{attribute 'OPC.UA.DA' := '1'}
FUNCTION_BLOCK EvosensLight EXTENDS LightBase
VAR_INPUT
END_VAR
VAR_OUTPUT
END_VAR
VAR
	{attribute 'OPC.UA.DA' := '0'}
	_config : EvosensLightConfig;	
	{attribute 'OPC.UA.DA' := '0'}
	_coeAccess : CoeAccess;	
	{attribute 'OPC.UA.DA' := '0'}
	_initConfigSerialCom : BOOL;	
	{attribute 'OPC.UA.DA' := '0'}
	_suffix : STRING := Const.CR_LF;
	{attribute 'OPC.UA.DA' := '0'}
	_serialCom  : SerialCom(Prefix :='', Suffix := _suffix);
	{attribute 'OPC.UA.DA' := '0'}
	_refSerialCom : REFERENCE TO SerialCom(Prefix :='', Suffix := _suffix) := _serialCom;		 
	{attribute 'OPC.UA.DA' := '0'}
	_isReceived : BOOL;
	
	{attribute 'OPC.UA.DA' := '0'}
	_deliverMessages : INT;
		
	StatusMsg : STRING(255);
	SwitchOnMsg : STRING(255);
	PowerMsg : STRING(255);
	IntensityMsg : STRING(255);	
	TemperatureMsg : STRING(255);
	LightSourcesMsg : STRING(255);
	TimeLightSourceMsg  : STRING(255);
	CustomMsg : STRING(255);
		
	{region 'Commands'}
	
	{attribute 'OPC.UA.DA' := '0'}
	_setSwitchOnCmd : BOOL;
	{attribute 'OPC.UA.DA' := '0'}
	_getSwitchOnCmd : BOOL;
	{attribute 'OPC.UA.DA' := '0'}
	_setPowerCmd : BOOL;
	{attribute 'OPC.UA.DA' := '0'}
	_getPowerCmd : BOOL;
	{attribute 'OPC.UA.DA' := '0'}
	_setIntensityCmd : BOOL;
	{attribute 'OPC.UA.DA' := '0'}
	_getIntensityCmd : BOOL;
	{attribute 'OPC.UA.DA' := '0'}
	_getTimeLightSourceCmd : BOOL;
	{attribute 'OPC.UA.DA' := '0'}
	_getLightSourcesCmd : BOOL;
	{attribute 'OPC.UA.DA' := '0'}
	_customCmd : BOOL;
	{attribute 'OPC.UA.DA' := '0'}			  		   
	_raisePropertiesCmd : BOOL;
	
	{attribute 'OPC.UA.DA' := '0'}
	_lightId : UINT; 
	{attribute 'OPC.UA.DA' := '0'}
	_switchOn : BOOL;
	{attribute 'OPC.UA.DA' := '0'}
	_setPower : LREAL;
	{attribute 'OPC.UA.DA' := '0'}
	_setIntensity : LREAL;
	{attribute 'OPC.UA.DA' := '0'}
	_cmd : STRING;	
		 
	{endregion}			
	
	{attribute 'OPC.UA.DA' := '0'}
	_initDevice : BOOL;	
	 
	{attribute 'OPC.UA.DA' := '0'}
	_lightSources : ARRAY [0..Const.PHOTOLUM_NUMBER_LIGHT_SOURCE] OF STRING(255);  
	
	{attribute 'OPC.UA.DA' := '0'}
	_itemScheduler : INT;
	{attribute 'OPC.UA.DA' := '0'}
	_itemInitScheduler : INT;
	{attribute 'OPC.UA.DA' := '0'}
	_itemExecScheduler : INT;		
	{attribute 'OPC.UA.DA' := '0'}
	_itemRaisedProperties : INT;			
	{attribute 'OPC.UA.DA' := '0'}
	_pulseGenerator : TON;	
	{attribute 'OPC.UA.DA' := '0'}
	_initPulseGenerator : TON;	
	{attribute 'OPC.UA.DA' := '0'}	
	_execPulseGenerator : TON;	
	
	{attribute 'OPC.UA.DA' := '0'}
	message : STRING;
	{attribute 'OPC.UA.DA' := '0'}
	lastMessage : STRING;	
	{attribute 'OPC.UA.DA' := '0'}
	sSubStr4 : STRING(4) := '';			
	{attribute 'OPC.UA.DA' := '0'}
	stringLength : INT;
	{attribute 'OPC.UA.DA' := '0'}
	_numberOfElements : DINT;
	{attribute 'OPC.UA.DA' := '0'}
	_indexNumberOfElements : INT;
END_VAR

IF NOT InitConfigSerialCom THEN
	ConfigureSerialCom();
ELSIF THIS^.Status = TExecutionState.Ready THEN
	SUPER^();	

	IF _refSerialCom.ErrorReceiveId = COMERROR_NOERROR THEN
		_refSerialCom(TxBuffer:= HardwareGlobalVariables.TxBufferLight, 
		 	      	  RxBuffer:= HardwareGlobalVariables.RxBufferLight);
	END_IF				  
	
	// Init device
	InitDevice(); 				  				 	
	
	IF StateMsg <> ANY_TO_STRING(State) THEN
		StateMsg := ANY_TO_STRING(State);
	END_IF
	
	// Deliver messages
	IF _refSerialCom.IsReceived THEN	
		lastMessage := _refSerialCom.LastReceivedString;			
		stringLength := LEN(lastMessage);
		
		IF stringLength > 2 THEN
			message := LEFT(lastMessage, stringLength - 2);
		ELSE
			message := ' ';
		END_IF; 	
			
		CASE _deliverMessages OF			
			EFeedbackMsgArduinoLight.SwitchOnMsg :
				SwitchOnMsg := message;	
			EFeedbackMsgArduinoLight.PowerMsg :
				PowerMsg := message;	
			EFeedbackMsgArduinoLight.IntensityMsg :
				IntensityMsg := message;	
			EFeedbackMsgArduinoLight.TemperatureMsg :
				TemperatureMsg := message;	
			EFeedbackMsgArduinoLight.LightSourcesMsg :
				LightSourcesMsg := message;			
				_logger.Information(_message.Reset().Append('LightSourcesMsg: ').Append(LightSourcesMsg).ToString());	
			EFeedbackMsgArduinoLight.TimeLightSourceMsg :
				TimeLightSourceMsg := message;	
			EFeedbackMsgArduinoLight.CustomMsg :
				CustomMsg := message;	
		END_CASE
	
		_deliverMessages := 0;
	END_IF								   							   	
		
	SetSwitchOn(_setSwitchOnCmd, TO_STRING(_lightId), _switchOn); 
	GetSwitchOn(_getSwitchOnCmd, TO_STRING(_lightId));
	SetPower(_setPowerCmd, TO_STRING(_lightId), _setPower);
	GetPower(_getPowerCmd, TO_STRING(_lightId));
	//SetIntensity(_setIntensityCmd, TO_STRING(_lightId), _setIntensity);
	//GetIntensity(_getIntensityCmd, TO_STRING(_lightId));
	GetTimeLightSource(_getTimeLightSourceCmd, TO_STRING(_lightId));
	GetLightSources(_getLightSourcesCmd);
	CustomCommand(_customCmd, _cmd);
	RaisePropertiesChanged(_raisePropertiesCmd, TO_STRING(_lightId));
	
	IF _initDevice AND NOT _setSwitchOnCmd AND NOT _getSwitchOnCmd AND NOT _setPowerCmd AND NOT _getPowerCmd AND NOT _setIntensityCmd AND NOT _getIntensityCmd
	   AND NOT _getTimeLightSourceCmd AND NOT _getLightSourcesCmd AND NOT _customCmd AND NOT _raisePropertiesCmd THEN
		MessageScheduler();
	END_IF
END_IF

METHOD ConfigureSerialCom
VAR_INPUT
END_VAR
IF _coeAccess.CoeOperation.Ready THEN
	_logger.Information(_message.Reset().Append('Start configuration com serial').ToString());
END_IF;	

_coeAccess.CoeOperation.Start();
_coeAccess(SerialCommunication := _config.SerialCommunication);
	
IF _coeAccess.CoeOperation.Done THEN
	_coeAccess.SetDone();	
	
	_Logger.Information(_message.Reset().
							Append('{').Append(TO_STRING(THIS^.Family)).Append('} : ').
							Append(' - Status : ').Append(TO_STRING(_coeAccess.Status)).ToString());	
	InitConfigSerialCom := TRUE;
END_IF
 
IF _coeAccess.CoeOperation.Error THEN	
	_coeAccess.SetError(0);
	
	_Logger.Error(_message.Reset().
							Append('{').Append(TO_STRING(THIS^.Family)).Append('} : ').
							Append(' - Status : ').Append(TO_STRING(_coeAccess.Status)).ToString());
	InitConfigSerialCom := TRUE;
END_IF

THIS^.Status := _coeAccess.Status;
State := _coeAccess.Status;
END_METHOD

{attribute 'TcRpcEnable' := '1'}
(** Custom command **)
METHOD CustomCommand
VAR_INPUT
	Execute : BOOL;
	Cmd : STRING;
END_VAR
IF Execute THEN
	_logger.Information(_message.Reset().Append(_config.Name).Append(' - Custom command : ').Append(Cmd).ToString());	
	_deliverMessages := EFeedbackMsgArduinoLight.CustomMsg;														
	_serialCom.Send(Cmd);	
	_customCmd := FALSE;
END_IF
END_METHOD

METHOD FB_init : BOOL
VAR_INPUT
	bInitRetains : BOOL; // if TRUE, the retain variables are initialized (warm start / cold start)
	bInCopyCode : BOOL;  // if TRUE, the instance afterwards gets moved into the copy code (online change)
	Config : EvosensLightConfig;
END_VAR
IF Config.IsEnabled THEN
	_config := Config;
	
	SUPER^._lightConfig.Name := Config.Name;
	SUPER^._lightConfig.DeviceID := Config.DeviceID;
	SUPER^._lightConfig.IsEnabled := Config.IsEnabled;
	SUPER^._lightConfig.LogLevel := Config.LogLevel;
	
	SUPER^.Name := Config.Name;
	SUPER^.DeviceID := Config.DeviceID;	
	THIS^.Family := DeviceFamily.Light;
		
	_Logger.Information(_message.Reset().Append('Init ').
							Append('{').Append(TO_STRING(THIS^.Family)).Append('} - ').
							Append('{').Append(TO_STRING(Config.Name)).Append('}').ToString());																													
END_IF
END_METHOD

{attribute 'TcRpcEnable' := '1'}
METHOD GetIntensity
VAR_INPUT
	Execute : BOOL;
	LightId : STRING;
END_VAR
VAR
	cmd : STRING := '*amps ';
END_VAR
IF Execute THEN	
	_deliverMessages := EFeedbackMsgArduinoLight.IntensityMsg;
	_serialCom.Send(CONCAT(cmd, LightId));
	
	_getIntensityCmd := FALSE;
END_IF
END_METHOD

METHOD GetLightSources
VAR_INPUT
	Execute: BOOL;
END_VAR
VAR
	cmd : STRING := '*light';
END_VAR
IF Execute THEN
	_logger.Information(_message.Reset().Append(_config.Name).Append(' - GetLightSources').ToString());
	_deliverMessages := EFeedbackMsgArduinoLight.LightSourcesMsg;
	_serialCom.Send(cmd);	
	
	_getLightSourcesCmd := FALSE;
END_IF
END_METHOD

{attribute 'TcRpcEnable' := '1'}
METHOD GetPower
VAR_INPUT
	Execute : BOOL;
	LightId : STRING;
END_VAR
VAR
	cmd : STRING := '*power ';
END_VAR
IF Execute THEN	
	_deliverMessages := EFeedbackMsgArduinoLight.PowerMsg;
	_serialCom.Send(CONCAT(cmd, LightId));
	
	 _getPowerCmd := FALSE;
END_IF
END_METHOD

{attribute 'TcRpcEnable' := '1'}
METHOD GetSwitchOn
VAR_INPUT
	Execute : BOOL;
	LightId : STRING;
END_VAR
VAR
	cmd : STRING := '*switch ';
END_VAR
IF Execute THEN	
	_deliverMessages := EFeedbackMsgArduinoLight.SwitchOnMsg;
	_serialCom.Send(CONCAT(cmd, LightId));
				
	_getSwitchOnCmd := FALSE;	
END_IF
END_METHOD

METHOD GetTemperature
VAR_INPUT
	LightId : STRING;
END_VAR
VAR
	cmd : STRING := '*temp ';
END_VAR
_deliverMessages := EFeedbackMsgArduinoLight.TemperatureMsg;
_serialCom.Send(CONCAT(cmd, LightId));
END_METHOD

METHOD GetTimeLightSource
VAR_INPUT
	Execute: BOOL;
	LightId : STRING;
END_VAR
VAR
	cmd : STRING := '*time ';
END_VAR
IF Execute THEN
	_logger.Information(_message.Reset().Append(_config.Name).Append(' - GetTimeLightSource - ').Append(LightId).ToString());
	_deliverMessages := EFeedbackMsgArduinoLight.TimeLightSourceMsg;
	_serialCom.Send(CONCAT(cmd, LightId));	
	
	_getTimeLightSourceCmd := FALSE;
END_IF
END_METHOD

PROPERTY InitConfigSerialCom : BOOL
GET
InitConfigSerialCom := _initConfigSerialCom;
END_GET
SET
_initConfigSerialCom := InitConfigSerialCom;
END_SET
END_PROPERTY

METHOD InitDevice
VAR_INPUT
END_VAR
VAR
	numElements : INT := 0;
    commaPos : INT;
    tempStr : STRING; 
	Separator : STRING := ',';
END_VAR
IF NOT _initDevice THEN	
	IF _initPulseGenerator.Q THEN
		_initPulseGenerator(IN := FALSE, PT := T#10MS);
			
		CASE _itemInitScheduler OF					
			0:	_logger.Information(_message.Reset().Append(_config.Name).Append(' - Init device').ToString());
				//_getLightSourcesCmd := TRUE;
				_itemInitScheduler := 50;
			
			1:	IF LightSourcesMsg <> '' THEN				
					tempStr := LightSourcesMsg;
					WHILE (LEN(tempStr) > 0) DO
						commaPos := FIND(tempStr, Separator);
						IF commaPos > 0 THEN
							_lightSources[numElements] := LEFT(tempStr, commaPos - 1);						
							tempStr := RIGHT(tempStr, LEN(tempStr) - commaPos);
						ELSE
							_lightSources[numElements] := tempStr;
							tempStr := ''; 
						END_IF
						_logger.Information(_message.Reset().Append(_config.Name).Append(' - ').Append(TO_STRING(numElements)).Append(': ').Append(_lightSources[numElements]).ToString());
						numElements := numElements + 1;						
					END_WHILE
														
					IF (numElements - 1) <> 0 THEN
						_numberOfElements := numElements;
						//_itemInitScheduler := 10; GVA
						_itemInitScheduler := 50;
					ELSE
						_itemInitScheduler := 40;	
					END_IF				
					
					_deliverMessages := -1;
				END_IF
			
			10: IF (_indexNumberOfElements >= 0) AND (_indexNumberOfElements < _numberOfElements) THEN
					tempStr := CONCAT(_lightSources[_indexNumberOfElements], ' 0');
					_serialCom.Send(CONCAT('*power ', tempStr));				
					_logger.Information(_message.Reset().Append(_config.Name).Append(' - ').Append(_lightSources[_indexNumberOfElements]).Append(' - Power: 0').ToString());	
					_indexNumberOfElements := _indexNumberOfElements + 1;
					
				ELSE
					_indexNumberOfElements := 0;
					_itemInitScheduler := 11;					
				END_IF	
			
			11: IF (_indexNumberOfElements >= 0) AND (_indexNumberOfElements < _numberOfElements) THEN
					tempStr := CONCAT(_lightSources[_indexNumberOfElements], ' 1');
					_serialCom.Send(CONCAT('*swit ', tempStr));
					_logger.Information(_message.Reset().Append(_config.Name).Append(' - ').Append(_lightSources[_indexNumberOfElements]).Append(' - Switch ON').ToString());
					_indexNumberOfElements := _indexNumberOfElements + 1;					
				ELSE
					_indexNumberOfElements := 0;
					_itemInitScheduler := 50;
				END_IF	

			41: _logger.Error(_message.Reset().Append(_config.Name).Append(' - numElements is empty: ').ToString());
				_itemInitScheduler := 50;	
		
			50: _initDevice := TRUE;
				_itemInitScheduler := 0;	
				_logger.Information(_message.Reset().Append(_config.Name).Append(' - Init device done').ToString());	
		END_CASE
	ELSE
		_initPulseGenerator(IN := TRUE, PT := T#100MS);		
	END_IF	
END_IF
END_METHOD

METHOD MessageScheduler
VAR_INPUT
END_VAR
VAR
	
END_VAR
IF _pulseGenerator.Q THEN
	_pulseGenerator(IN := FALSE, PT := T#10MS);
		
	CASE _itemScheduler OF					
		0:	_getSwitchOnCmd := TRUE;
			_itemScheduler := 1;
			
		1:	_getPowerCmd := TRUE;
			_itemScheduler := 2;
			
		2:  //GetTemperature(_lightID);			
			_itemScheduler := 10;
			
		10: IF _lightId > 0 AND _lightId < Const.PHOTOLUM_NUMBER_LIGHT_SOURCE THEN
				_lightId := _lightId + 1;				
			ELSE
				_lightId := 1;
			END_IF
			
			
			_itemScheduler := 0;
									
	END_CASE
ELSE
	_pulseGenerator(IN := TRUE, PT := T#250MS);		
END_IF


IF _pulseIsAliveGenerator.Q THEN
	_pulseIsAliveGenerator(IN := FALSE, PT := T#10MS);
		
	IsAlive();	
ELSE
	_pulseIsAliveGenerator(IN := TRUE, PT := T#1000MS);		
END_IF
END_METHOD

{attribute 'TcRpcEnable' := '1'}
METHOD RaisePropertiesChanged
VAR_INPUT
	Execute : BOOL;
	LightId : STRING;
END_VAR
VAR
	numElements : INT := 0;
    commaPos : INT;
    tempStr : STRING; 
	Separator : STRING := ',';
END_VAR
IF Execute THEN
	_raisePropertiesCmd := TRUE;
	IF LightId <> '' THEN
		_lightId := STRING_TO_UINT(LightId);
	END_IF
	
	IF _pulseGenerator.Q THEN
		_pulseGenerator(IN := FALSE, PT := T#10MS);	

		CASE _itemRaisedProperties OF
			0:  SwitchOnMsg := ' ';
				PowerMsg := ' ';		
				IntensityMsg := ' ';
				LightSourcesMsg := ' ';		
				TimeLightSourceMsg := ' ';		
				_itemRaisedProperties := 1;					

			1:  IF _lightId > 0 AND _lightId <= Const.PHOTOLUM_NUMBER_LIGHT_SOURCE THEN
					_itemRaisedProperties := 50;	
				ELSE
					_itemRaisedProperties := 40;	
				END_IF  
				
			10: _getSwitchOnCmd := TRUE;													
				_itemRaisedProperties := 11;
				
			11: IF SwitchOnMsg <> ' ' THEN
					_itemRaisedProperties := 12;
				END_IF	
				
			12: _getPowerCmd := TRUE;													
				_itemRaisedProperties := 13;
				
			13: IF PowerMsg <> ' ' THEN
					_itemRaisedProperties := 16;
				END_IF
							
			16: _getTimeLightSourceCmd := TRUE;													
				_itemRaisedProperties := 17;
				
			17: IF TimeLightSourceMsg <> ' ' THEN
					_itemRaisedProperties := 50;
				END_IF
			
			40: _logger.Error(_message.Reset().Append(_config.Name).Append(' - RaisePropertiesChanged - LightId is empty').ToString());
				_itemRaisedProperties := 50;
			
			50:  _logger.Information(_message.Reset().Append(_config.Name).Append(' - RaisePropertiesChanged').ToString());
				_raisePropertiesCmd := FALSE;				
				_itemRaisedProperties := 0;
			
		END_CASE
	ELSE
		_pulseGenerator(IN := TRUE, PT := T#100MS);	
	END_IF
END_IF
END_METHOD

{attribute 'TcRpcEnable' := '1'}
METHOD SetIntensity
VAR_INPUT
	Execute : BOOL;
	LightId : STRING;
	Intensity : LREAL;
END_VAR
VAR
	cmd : STRING := '*amps ';
	tmpConcatLightIdIntensity : STRING;
END_VAR
IF Execute THEN	
	_setIntensityCmd := TRUE;
	_setIntensity := Intensity; 
	IF LightId <> '' THEN
		_lightId := STRING_TO_UINT(LightId);
	END_IF
	
	IF _execPulseGenerator.Q THEN
		_execPulseGenerator(IN := FALSE, PT := T#10MS);
			
		CASE _itemExecScheduler OF
			0:  IF _lightId > 0 AND _lightId <= Const.PHOTOLUM_NUMBER_LIGHT_SOURCE THEN
					_itemExecScheduler := 10;	
				ELSE
					_itemExecScheduler := 40;	
				END_IF
				
				_deliverMessages := -1;

			10: tmpConcatLightIdIntensity := CONCAT(CONCAT(TO_STRING(_lightId), ' '), TO_STRING(Intensity));

				_logger.Information(_message.Reset().Append(_config.Name).Append(' - ').Append(TO_STRING(_lightId)).Append(' - SetIntensity : ').Append(TO_STRING(_lightId)).Append(' - ').Append(TO_STRING(Intensity)).ToString());
				_serialCom.Send(CONCAT(cmd, TO_STRING(tmpConcatLightIdIntensity)));
				_itemExecScheduler := 11;
			
			11:  _getIntensityCmd := TRUE;
				_itemExecScheduler := 50;
			
			40: _logger.Error(_message.Reset().Append(_config.Name).Append(' - SetIntensity - light id is not valid').ToString());
				_itemExecScheduler := 50;
		
			50:  _setIntensityCmd := FALSE;	
				_itemExecScheduler := 0;		
								
		END_CASE
	ELSE
		_execPulseGenerator(IN := TRUE, PT := T#100MS);	
	END_IF
END_IF
END_METHOD

{attribute 'TcRpcEnable' := '1'}
METHOD SetPower
VAR_INPUT
	Execute : BOOL;
	LightId : STRING;
	Power : LREAL;
END_VAR
VAR
	cmd : STRING := '*power ';
	tmpConcatLightIdPower : STRING;
END_VAR
IF Execute THEN	
	_setPowerCmd := TRUE;		
	_setPower := Power;	
	IF LightId <> '' THEN
		_lightId := STRING_TO_UINT(LightId);
	END_IF
	
	IF _execPulseGenerator.Q THEN
		_execPulseGenerator(IN := FALSE, PT := T#10MS);
			
		CASE _itemExecScheduler OF
			0: IF _lightId > 0 AND _lightId <= Const.PHOTOLUM_NUMBER_LIGHT_SOURCE THEN
					_itemExecScheduler := 10;	
				ELSE
					_itemExecScheduler := 40;	
				END_IF
				
				_deliverMessages := -1;

			10: tmpConcatLightIdPower := CONCAT(CONCAT(TO_STRING(_lightId), ' '), TO_STRING(Power));

				_logger.Information(_message.Reset().Append(_config.Name).Append(' - ').Append(TO_STRING(_lightId)).Append(' - SetPower : ').Append(TO_STRING(Power)).ToString());
				_serialCom.Send(CONCAT(cmd, TO_STRING(tmpConcatLightIdPower)));
				_itemExecScheduler := 11;
			
			11:  _getPowerCmd := TRUE;
				_itemExecScheduler := 50;
			
			40: _logger.Error(_message.Reset().Append(_config.Name).Append(' - SetPower - light id is not valid').ToString());
				_itemExecScheduler := 50;
	
			50:  _setPowerCmd := FALSE;	
				_itemExecScheduler := 0;		
								
		END_CASE
	ELSE
		_execPulseGenerator(IN := TRUE, PT := T#100MS);	
	END_IF
END_IF
END_METHOD

{attribute 'TcRpcEnable' := '1'}
METHOD SetSwitchOn
VAR_INPUT
	Execute : BOOL;	
	LightId : STRING;
	SwitchOn : BOOL;
END_VAR
VAR
	cmd : STRING := '*switch ';
	tmpConcatLightIdSwitchOn : STRING;
	tmp : STRING;
	switchOnValue : STRING;
END_VAR
IF Execute THEN	
	_setSwitchOnCmd := TRUE;	
	_switchOn := SwitchOn; 
	
	IF LightId <> '' THEN
		_lightId := STRING_TO_UINT(LightId);
	END_IF	
	
	IF _execPulseGenerator.Q THEN
		_execPulseGenerator(IN := FALSE, PT := T#10MS);
			
		CASE _itemExecScheduler OF
			0:  IF _lightId > 0 AND _lightId <= Const.PHOTOLUM_NUMBER_LIGHT_SOURCE THEN
					_itemExecScheduler := 10;	
				ELSE
					_itemExecScheduler := 40;	
				END_IF
				
				_deliverMessages := -1;

			10:	IF _switchOn THEN
					switchOnValue := 'ON';
				ELSE
					switchOnValue := 'OFF';
				END_IF
				tmpConcatLightIdSwitchOn := CONCAT(CONCAT(TO_STRING(_lightId), ' '), TO_STRING(switchOnValue));
				
				_logger.Information(_message.Reset().Append(_config.Name).Append(' - ').Append(TO_STRING(_lightId)).Append(' - SwitchOn : ').Append(TO_STRING(switchOnValue)).ToString());
				tmp := CONCAT(cmd, TO_STRING(tmpConcatLightIdSwitchOn));
				_serialCom.Send(tmp);
				_itemExecScheduler := 11;
			
			11:  _getSwitchOnCmd := TRUE;
				_itemExecScheduler := 50;
				
			40: _logger.Error(_message.Reset().Append(_config.Name).Append(' - SwitchOn - light id is not valid').ToString());
				_itemExecScheduler := 50;
				
			50:  _setSwitchOnCmd := FALSE;	
				_switchOn := FALSE;
				_itemExecScheduler := 0;		
								
		END_CASE
	ELSE
		_execPulseGenerator(IN := TRUE, PT := T#200MS);	
	END_IF
END_IF
END_METHOD

END_FUNCTION_BLOCK

(* stored: Version 1.1.0.1, ProductVersion 3.1.4024.12
   POU EvosensLight: Id {6cd5921a-4584-4484-a5b0-4ceb6ba5fa9c}, SpecialFunc None
   Folder Commands: Id {c9612207-3069-403a-a008-7feb6fbcaaa1}
   Method ConfigureSerialCom: Id {ff46e15c-5e1b-4515-aedc-4bda88b9b543}
   Method CustomCommand: Id {1c035ed9-e5e3-4cb2-a1c3-745927324251}
   Method FB_init: Id {c91c8837-368d-495f-8bb2-f6da283d6563}
   Method GetIntensity: Id {0457c760-e12a-4227-946a-1470c71c278d}
   Method GetLightSources: Id {6ccfe94b-96b4-4231-9e24-54e630f85ff3}
   Method GetPower: Id {2008567d-8399-4be1-bc97-207de4b206c4}
   Method GetSwitchOn: Id {a038a969-dedb-4742-92c2-c2c03b015813}
   Method GetTemperature: Id {bfd539f6-71b0-40cf-b880-46ee8a0e89c7}
   Method GetTimeLightSource: Id {0495df94-72fa-4aec-810e-4f5e006ea259}
   Property InitConfigSerialCom: Id {de09a242-23e0-4081-80ba-03ae9084e36b}
   Get Get: Id {80c46679-8f6b-457f-8777-817f707cd876}
   Set Set: Id {4c46eeed-2bfd-4b1a-9888-39860f1d007f}
   Method InitDevice: Id {2e39d23c-210a-4982-a0ad-5d282f1f053b}
   Method MessageScheduler: Id {6e9229aa-2d7b-4bca-b16d-bc3397c7fe77}
   Method RaisePropertiesChanged: Id {19738d45-1f97-44b5-bfde-85a52063c67f}
   Method SetIntensity: Id {70b75109-6226-4822-a750-5a38c8c0bd07}
   Method SetPower: Id {bd091d4f-20c8-47b0-8f95-d76a242455e4}
   Method SetSwitchOn: Id {27eda15d-e9db-4eeb-99e6-1ab9f7ad7825} *)
